// TIA Portal V17 export
// export: Created 2022-07-20T07:02:34.4826547Z, ExportSetting WithDefaults, DisplayName Totally Integrated Automation Portal, DisplayVersion V17, DisplayName TIA Portal Openness, DisplayVersion V17, DisplayName TIA Portal Version Control Interface, DisplayVersion V17, DisplayName SINAMICS Startdrive Advanced, DisplayVersion V17, DisplayName SINAMICS Startdrive G130, G150, S120, S150, SINAMICS MV, S210, DisplayVersion V17, DisplayName SINAMICS Startdrive G110M, G120, G120C, G120D, G120P, G115D, DisplayVersion V17, DisplayName STEP 7 Professional, DisplayVersion V17, DisplayName STEP 7 Safety, DisplayVersion V17, DisplayName WinCC Advanced, DisplayVersion V17
FUNCTION_BLOCK "FB10371_IOLinkConfig_DV2121"   // FB10371, LAD
{ S7_Optimized_Access := 'TRUE' }
VERSION : 0.1
// stored: AutoNumber false, IsIECCheckEnabled false, IsRetainMemResEnabled false, MemoryReserve 100, SetENOAutomatically false, UDAEnableTagReadback false
   VAR_INPUT
      Ackowledge : Bool;
      PortDevice : Int;
      Id : HW_IO;
      RequestResetDefaultSettings : Bool;
      RequestTeachSP1 : Bool;
      RequestTeachSP2 : Bool;
      RequestPowerCycles : Bool;
      RequestParamConfigFault : Bool;
      RequestOperatingHours : Bool;
      SP1_Value : Bool;
   END_VAR
   VAR_OUTPUT
      ResetDefaultSettingsDone : Bool;
      TeachSP1Done : Bool;
      TeachSP2Done : Bool;
      PowerCycleReadingDone : Bool;
      OperatingHourReadingDone : Bool;
      ParamConfigReadingdone : Bool;
      NumberOfCycles : UInt;
      NumberOfHours : UInt;
      ParamConfigFault : Array[0..231] of Byte;
      Error : Bool;
      Status : Word;
   END_VAR
   VAR
      CommandStruct : Struct
         In : Struct
            TrigStart_Pulse : Bool;
            Id : HW_IO;
            rw : Bool;
            Port : Int;
            index : Int;
            subindex : Int;
            length : Int;
         END_STRUCT;
         Out : Struct
            Done : Bool;
            busy : Bool;
            Error : Bool;
            Status : Word;
         END_STRUCT;
         InOut : Struct
            Data : Array[0..231] of Byte;
         END_STRUCT;
      END_STRUCT;
      RequestPulseTrigStart : Bool;
      IoLinkConfigurationStateDiagram : Int;
      ParameterDone : Bool;
      R_TRIG_RequestResetDefautSettings : R_TRIG;
      R_TRIG_RequestTeachSP1 { S7_SetPoint := 'True'} : R_TRIG;
      R_TRIG_RequestTeachSP2 { S7_SetPoint := 'True'} : R_TRIG;
      R_TRIG_RequestPowerCycles { S7_SetPoint := 'True'} : R_TRIG;
      R_TRIG_RequestOperatingHours { S7_SetPoint := 'True'} : R_TRIG;
      R_TRIG_RequestParamConfigFault { S7_SetPoint := 'True'} : R_TRIG;
      FB10003_Pulse_Instance { S7_SetPoint := 'True'} : "FB10003_Pulse";
      FB10370_IoLinkDevice_Instance_1 { S7_SetPoint := 'True'} : "FB10370_IoLinkDevice";
   END_VAR
   VAR CONSTANT
      WAIT_FOR_IO_LINK_CONFIGURATION_COMMAND : Int := 0;
      RESTORE_DEFAULT_SETTINGS_IN_PROGRESS : Int := 10;
      TEACH_SP1_IN_PROGRESS : Int := 20;
      TEACH_SP2_IN_PROGRESS : Int := 30;
      READ_POWER_CYCLES_IN_PROGRESS : Int := 40;
      READ_OPERATING_HOURS_IN_PROGRESS : Int := 50;
      READ_PARAM_CONFIG_FAULT_IN_PROGRESS : Int := 60;
      IO_LINK_COMMAND_CONFIGURATION_DONE : Int := 100;
      CAP_IO_LINK_IFM : Int := 19456;
   END_VAR
BEGIN

REGION Network 1 (SCL): First Scan
   IF "FirstScan" THEN
       #ResetDefaultSettingsDone := FALSE;
       #TeachSP1Done := FALSE;
       #IoLinkConfigurationStateDiagram := #WAIT_FOR_IO_LINK_CONFIGURATION_COMMAND;
   END_IF;
END_REGION

REGION Network 2 (SCL): Edge Signals, Timers, Pulse
   REGION EDGE SIGNALS 
       #R_TRIG_RequestResetDefautSettings(CLK := #RequestResetDefaultSettings);
       #R_TRIG_RequestTeachSP1(CLK := #RequestTeachSP1);
       #R_TRIG_RequestTeachSP2(CLK := #RequestTeachSP2);
       #R_TRIG_RequestPowerCycles(CLK := #RequestPowerCycles);
       #R_TRIG_RequestOperatingHours(CLK := #RequestOperatingHours);
       #R_TRIG_RequestParamConfigFault(CLK := #RequestParamConfigFault);

   END_REGION

   REGION TIMERS 

   END_REGION

   REGION PULSE
       #FB10003_Pulse_Instance(CLK := #RequestPulseTrigStart,
                               PT := T#50ms,
                               Q := #CommandStruct.In.TrigStart_Pulse);
   END_REGION
END_REGION

REGION Network 3 (SCL): Io Link Commands Management
   #CommandStruct.In.Port := #PortDevice;
   #CommandStruct.In.Id := #Id;
END_REGION

REGION Network 4: Io Link Configuration Manager
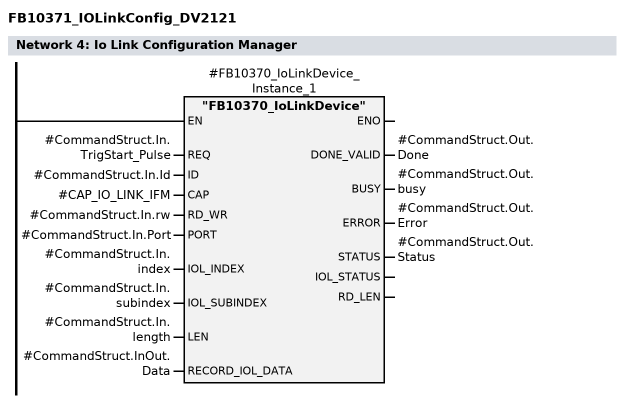
   RUNG wire#powerrail
      #FB10370_IoLinkDevice_Instance_1(REQ := #CommandStruct.In.TrigStart_Pulse, ID := #CommandStruct.In.Id, CAP := #CAP_IO_LINK_IFM, RD_WR := #CommandStruct.In.rw, PORT := #CommandStruct.In.Port, IOL_INDEX := #CommandStruct.In.index, IOL_SUBINDEX := #CommandStruct.In.subindex, LEN := #CommandStruct.In.length, RECORD_IOL_DATA := #CommandStruct.InOut.Data, DONE_VALID => #CommandStruct.Out.Done, BUSY => #CommandStruct.Out.busy, ERROR => #CommandStruct.Out.Error, STATUS => #CommandStruct.Out.Status, IOL_STATUS =>, RD_LEN =>)
   END_RUNG
   // the same network as SCL:
   #FB10370_IoLinkDevice_Instance_1(REQ := #CommandStruct.In.TrigStart_Pulse,   // "FB10370_IoLinkDevice"
                           ID := #CommandStruct.In.Id,
                           CAP := #CAP_IO_LINK_IFM,
                           RD_WR := #CommandStruct.In.rw,
                           PORT := #CommandStruct.In.Port,
                           IOL_INDEX := #CommandStruct.In.index,
                           IOL_SUBINDEX := #CommandStruct.In.subindex,
                           LEN := #CommandStruct.In.length,
                           RECORD_IOL_DATA := #CommandStruct.InOut.Data,
                           DONE_VALID => #CommandStruct.Out.Done,
                           BUSY => #CommandStruct.Out.busy,
                           ERROR => #CommandStruct.Out.Error,
                           STATUS => #CommandStruct.Out.Status);
END_REGION

REGION Network 5 (SCL): Io Link Commands Configuration Management
   CASE #IoLinkConfigurationStateDiagram OF

       #WAIT_FOR_IO_LINK_CONFIGURATION_COMMAND:
           IF #R_TRIG_RequestResetDefautSettings.Q THEN
               #ResetDefaultSettingsDone := FALSE;
               #CommandStruct.InOut.Data[0] := 10#130;
               IF #ParameterDone THEN
                   #IoLinkConfigurationStateDiagram := #RESTORE_DEFAULT_SETTINGS_IN_PROGRESS;
               END_IF;
           ELSIF #R_TRIG_RequestTeachSP1.Q THEN
               #TeachSP1Done := FALSE;
               #CommandStruct.InOut.Data[0] := 10#65;
               IF #ParameterDone THEN
                   #IoLinkConfigurationStateDiagram := #TEACH_SP1_IN_PROGRESS;
               END_IF;
           ELSIF #R_TRIG_RequestTeachSP2.Q THEN
               #TeachSP1Done := FALSE;
               #CommandStruct.InOut.Data[0] := 10#66;
               IF #ParameterDone THEN
                   #IoLinkConfigurationStateDiagram := #TEACH_SP2_IN_PROGRESS;
               END_IF;
           ELSIF #R_TRIG_RequestPowerCycles.Q THEN
               #PowerCycleReadingDone := FALSE;
               IF #ParameterDone THEN
                   #IoLinkConfigurationStateDiagram := #READ_POWER_CYCLES_IN_PROGRESS;
               END_IF;
           ELSIF #R_TRIG_RequestOperatingHours.Q THEN
               #OperatingHourReadingDone := FALSE;
               IF #ParameterDone THEN
                   #IoLinkConfigurationStateDiagram := #READ_OPERATING_HOURS_IN_PROGRESS;
               END_IF;
           ELSIF #R_TRIG_RequestParamConfigFault.Q THEN
               #ParamConfigReadingdone := FALSE;
               IF #ParameterDone THEN
                   #IoLinkConfigurationStateDiagram := #READ_PARAM_CONFIG_FAULT_IN_PROGRESS;
               END_IF;
           END_IF;

       #RESTORE_DEFAULT_SETTINGS_IN_PROGRESS:
           REGION State Action Management
               #RequestPulseTrigStart := TRUE;
           END_REGION

           REGION State Exit Management
               IF #CommandStruct.Out.Done THEN
                   #ResetDefaultSettingsDone := TRUE;
                   #RequestPulseTrigStart := FALSE;
                   #CommandStruct.In.rw := FALSE;
                   #IoLinkConfigurationStateDiagram := #IO_LINK_COMMAND_CONFIGURATION_DONE;
               END_IF;
           END_REGION

       #TEACH_SP1_IN_PROGRESS:
           REGION State Action Management
               #RequestPulseTrigStart := TRUE;
              // #CommandStruct.In.Data := #SP1_Value;
           END_REGION

           REGION State Exit Management
               IF #CommandStruct.Out.Done THEN
                   #TeachSP1Done := TRUE;
                   #RequestPulseTrigStart := FALSE;
                   #IoLinkConfigurationStateDiagram := #IO_LINK_COMMAND_CONFIGURATION_DONE;
               END_IF;
           END_REGION

       #TEACH_SP2_IN_PROGRESS:
           REGION State Action Management
               #RequestPulseTrigStart := TRUE;
               // #CommandStruct.In.Data := #SP1_Value;
           END_REGION

           REGION State Exit Management
               IF #CommandStruct.Out.Done THEN
                   #TeachSP1Done := TRUE;
                   #RequestPulseTrigStart := FALSE;
                   #IoLinkConfigurationStateDiagram := #IO_LINK_COMMAND_CONFIGURATION_DONE;
               END_IF;
           END_REGION

       #READ_POWER_CYCLES_IN_PROGRESS:
           REGION State Action Management
               #RequestPulseTrigStart := TRUE;
               // #CommandStruct.In.Data := #SP1_Value;
           END_REGION

           REGION State Exit Management
               IF #CommandStruct.Out.Done THEN
                   #NumberOfCycles := UDINT_TO_UINT("FC10330_2BytesToUDint"(LowByte := #CommandStruct.InOut.Data[0], HighByte := #CommandStruct.InOut.Data[1]));               
                   #PowerCycleReadingDone := TRUE;
                   #RequestPulseTrigStart := FALSE;
                   #IoLinkConfigurationStateDiagram := #IO_LINK_COMMAND_CONFIGURATION_DONE;
               END_IF;
           END_REGION

       #READ_OPERATING_HOURS_IN_PROGRESS:
           REGION State Action Management
               #RequestPulseTrigStart := TRUE;
               // #CommandStruct.In.Data := #SP1_Value;
           END_REGION

           REGION State Exit Management
               IF #CommandStruct.Out.Done THEN
                   #NumberOfHours := UDINT_TO_UINT("FC10330_2BytesToUDint"(LowByte := #CommandStruct.InOut.Data[0], HighByte := #CommandStruct.InOut.Data[1]));
                   #PowerCycleReadingDone := TRUE;
                   #RequestPulseTrigStart := FALSE;
                   #IoLinkConfigurationStateDiagram := #IO_LINK_COMMAND_CONFIGURATION_DONE;
               END_IF;
           END_REGION

       #READ_PARAM_CONFIG_FAULT_IN_PROGRESS:
           REGION State Action Management
               #RequestPulseTrigStart := TRUE;
               // #CommandStruct.In.Data := #SP1_Value;
           END_REGION

           REGION State Exit Management
               IF #CommandStruct.Out.Done THEN
                   #ParamConfigFault := #CommandStruct.InOut.Data;
                   #ParamConfigReadingdone := TRUE;
                   #RequestPulseTrigStart := FALSE;
                   #IoLinkConfigurationStateDiagram := #IO_LINK_COMMAND_CONFIGURATION_DONE;
               END_IF;
           END_REGION
       #IO_LINK_COMMAND_CONFIGURATION_DONE:
           #ParameterDone := FALSE;
           #IoLinkConfigurationStateDiagram := #WAIT_FOR_IO_LINK_CONFIGURATION_COMMAND;
   END_CASE;
END_REGION

REGION Network 6 (SCL): Io Link Commands Error Management
   IF #CommandStruct.Out.Error THEN
       #IoLinkConfigurationStateDiagram := #WAIT_FOR_IO_LINK_CONFIGURATION_COMMAND;
       #Error := TRUE;
   END_IF;

   IF #Ackowledge THEN
       #Error := FALSE;
   END_IF;
   #Status := #CommandStruct.Out.Status;
END_REGION

REGION Network 7 (SCL): Io Link Commands States Management
   IF #R_TRIG_RequestResetDefautSettings.Q OR #R_TRIG_RequestTeachSP1.Q OR #R_TRIG_RequestTeachSP2.Q THEN
       #CommandStruct.In.index:= 2;
       #CommandStruct.In.subindex:=0;
       #CommandStruct.In.rw := TRUE;
       #CommandStruct.In.length := 8;
       #ParameterDone := TRUE;
   ELSIF #R_TRIG_RequestPowerCycles.Q THEN
       #CommandStruct.In.index := 541;
       #CommandStruct.In.subindex := 0;
       #CommandStruct.In.rw := FALSE;
       #CommandStruct.In.length := 16;
       #ParameterDone := TRUE;
   ELSIF #R_TRIG_RequestOperatingHours.Q THEN
       #CommandStruct.In.index := 542;
       #CommandStruct.In.subindex := 0;
       #CommandStruct.In.rw := FALSE;
       #CommandStruct.In.length := 16;
       #ParameterDone := TRUE;
   ELSIF #R_TRIG_RequestParamConfigFault.Q THEN
       #CommandStruct.In.index := 546;
       #CommandStruct.In.subindex := 0;
       #CommandStruct.In.rw := FALSE;
       #CommandStruct.In.length := 16;
       #ParameterDone := TRUE;
   END_IF;
END_REGION
END_FUNCTION_BLOCK
